// TwinCAT 3 PLC project Git_TcProjectCompare_Test
// ProgramVersion: 3.1.4023.0
// libraries:
//   Tc2_Standard, * (Beckhoff Automation GmbH)
//   Tc2_System, * (Beckhoff Automation GmbH)
//   Tc3_Module, * (Beckhoff Automation GmbH)
// project tree:
//   / PlcTask.TcTTO
//   POUs/ FB_OtherThing.TcPOU, FB_TheThing.TcPOU, MAIN.TcPOU

CONFIGURATION Git_TcProjectCompare_Test
    RESOURCE PLC ON TwinCAT3
        TASK PlcTask(INTERVAL := T#10ms, PRIORITY := 20);
        PROGRAM MAIN WITH PlcTask : MAIN;
    END_RESOURCE
END_CONFIGURATION

// ---- POUs/MAIN.TcPOU
PROGRAM MAIN
VAR
	TheThing	: FB_TheThing;
	OtherThing	: FB_OtherThing;
END_VAR

thething();
IF theThing.prepare_to_do_the_thing() THEN
	theThing.do_the_thing();
END_IF

END_PROGRAM

// ---- POUs/FB_TheThing.TcPOU
FUNCTION_BLOCK FB_TheThing
VAR_INPUT
	input	: REAL;
END_VAR
VAR_OUTPUT
	output	: REAL;
END_VAR
VAR

	prepared			: BOOL := FALSE;
	succeeded			: BOOL := FALSE;
	
	preparation_timer	: TON;
	
	offset				: REAL := 0;
	testAdd				: BOOL;
	
END_VAR


prepared := prepare_to_do_the_thing();

succeeded := do_the_thing();

METHOD do_the_thing : BOOL
VAR_INPUT
END_VAR
THIS^.output := SEL(THIS^.prepared, 0, input - THIS^.offset);

do_the_thing := NOT THIS^.prepared;
END_METHOD

METHOD prepare_to_do_the_thing : BOOL
VAR_INPUT

END_VAR
preparation_timer(IN := NOT THIS^.prepared, PT := T#3S);

THIS^.offset := SEL(preparation_timer.Q, THIS^.offset, (THIS^.offset + input) / 2);

prepare_to_do_the_thing := NOT preparation_timer.Q;
END_METHOD

END_FUNCTION_BLOCK

// ---- POUs/FB_OtherThing.TcPOU
FUNCTION_BLOCK FB_OtherThing
VAR_INPUT
END_VAR
VAR_OUTPUT
END_VAR
VAR
	counter	: INT; 
END_VAR

counter := counter + 1

METHOD DoSomething : BOOL
VAR_INPUT
END_VAR
counter := counter + 1
END_METHOD

END_FUNCTION_BLOCK
